Omron Sysmac Studio project comodo-gateway_1.0 (Sysmac Studio 1.64.0.64008, StandardProject)

# Controller new_Controller_0: NX102-9020 version 1.50
Units and slaves: Unit 1 : NX-PF0730 (N1); Unit 2 : NX-ID4442 (N2); Unit 3 : NX-OD4256 (N3)
Task PrimaryTask (priority 4, period or condition 2000): Program0
Library comodo-sync-lib_abb 0.4.0 (contents left out)

VAR_GLOBAL
    Is_Monitoring : BOOL;  (* published *)
    Is_Moving_Linear : BOOL;  (* published *)
    Robot_Out : LWORD;  (* network input *)
    Robot_In : LWORD;  (* network output *)
    Robot_Positions : ARRAY[0..5] OF LREAL;
    In_Joint_1 : LREAL;  (* published *)
    In_Joint_2 : LREAL;  (* published *)
    In_Joint_3 : LREAL;  (* published *)
    In_Joint_4 : LREAL;  (* published *)
    In_Joint_5 : LREAL;  (* published *)
    In_Joint_6 : LREAL;  (* published *)
    Out_Joint_1 : LREAL;  (* published *)
    Out_Joint_2 : LREAL;  (* published *)
    Out_Joint_3 : LREAL;  (* published *)
    Out_Joint_4 : LREAL;  (* published *)
    Out_Joint_5 : LREAL;  (* published *)
    Out_Joint_6 : LREAL;  (* published *)
END_VAR

PROGRAM Program0
VAR
    ParseCurrentPosition : ParseRobotData;
END_VAR
VAR_EXTERNAL
    Is_Monitoring : BOOL;
END_VAR

(* Section Section0: ladder, written here as Structured Text *)

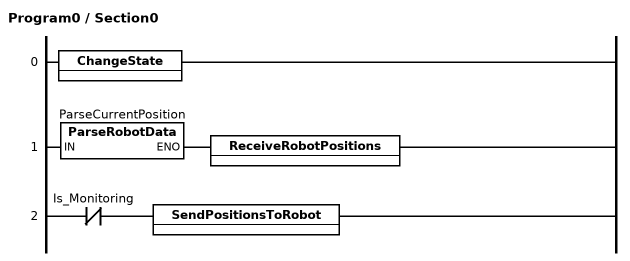
(* Rung 0 *)
(* Rung 1 *)
ParseCurrentPosition(IN := TRUE);
(* Rung 2 *)
(* drawn but driving nothing: Is_Monitoring *)
END_PROGRAM